FUNCTION_BLOCK FB_SlaveRobot
VAR
	// slave arms, responsible for arm kinematic and control
	m_slaveArms :ARRAY[1..g_sArmNum] OF FB_SlaveArm;
	
	// arm light control word
	m_lightCrlWord :ARRAY [1..4] OF UDINT;
	
	// arm state
	m_slaveArmState:ARRAY[1..g_sArmNum] OF E_SlaveArmState:=[g_sArmNum(E_SlaveArmState.SlaveArmState_Error)];
	m_lastSlaveArmState:ARRAY[1..g_sArmNum] OF E_SlaveArmState:=[g_sArmNum(E_SlaveArmState.SlaveArmState_Error)];
	m_nextSlaveArmState:ARRAY[1..g_sArmNum] OF E_SlaveArmState:=[g_sArmNum(E_SlaveArmState.SlaveArmState_Error)];
	
	// flag if panel and instrument mounted
	m_panelMountedFlag :ARRAY[1..g_sArmNum] OF BOOL :=[g_sArmNum(FALSE)];
	m_instrumentMountedFlag :ARRAY[1..g_sArmNum] OF BOOL :=[g_sArmNum(FALSE)];
	
	// all arm controller instance 
	m_armCtrlFactory :ARRAY[1..g_sArmNum,1..SlaveArmState_totalNum] OF I_SlaveArmCtrl;
	m_armError :ARRAY[1..g_sArmNum] OF FB_SlaveCtrlError;
	m_armInit :ARRAY[1..g_sArmNum] OF FB_SlaveCtrlInit;
	m_armSelfCheck :ARRAY[1..g_sArmNum] OF FB_SlaveCtrlSelfCheck;
	m_armStandBy :ARRAY[1..g_sArmNum] OF FB_SlaveCtrlStandBy;
	m_mountPanel :ARRAY[1..g_sArmNum] OF FB_SlaveCtrlMountPanel;
	m_panelReady :ARRAY[1..g_sArmNum] OF FB_SlaveCtrlPanelReady;
	m_mountInstru :ARRAY[1..g_sArmNum] OF FB_SlaveCtrlMountInstru;
	m_instruReady :ARRAY[1..g_sArmNum] OF FB_SlaveCtrlInstruReady;
	m_armMasterSlave :ARRAY[1..g_sArmNum] OF FB_SlaveCtrlMasterSlave;
	m_scopeReady :ARRAY[1..g_sArmNum] OF FB_SlaveCtrlScopeReady;
	m_armEndoscope :ARRAY[1..g_sArmNum] OF FB_SlaveCtrlEndoscope;
	m_armAdjust :ARRAY[1..g_sArmNum] OF FB_SlaveCtrlAdjust;
	m_armPackage :ARRAY[1..g_sArmNum] OF FB_SlaveCtrlPackage;
	m_armCart :ARRAY[1..g_sArmNum] OF FB_SlaveCtrlCart;
	m_armGraCali :ARRAY[1..g_sArmNum] OF FB_SlaveCtrlGraCali;
	m_armTest :ARRAY[1..g_sArmNum] OF FB_SlaveCtrlTest;
	m_instruRetract :ARRAY[1..g_sArmNum] OF FB_SlaveCtrlInstruRetract;
	m_instruInvasion :ARRAY[1..g_sArmNum] OF FB_SlaveCtrlInstruInvasion;
	m_armDisable :ARRAY[1..g_sArmNum] OF FB_SlaveCtrlDisable;
	m_instruCali :ARRAY[1..g_sArmNum] OF FB_SlaveCtrlInstruCali;
	m_scopeToggle :ARRAY[1..g_sArmNum] OF FB_SlaveCtrlScopeToggle;
	m_Performance :ARRAY[1..g_sArmNum] OF FB_SlaveCtrlPerformance;
	m_armStop :ARRAY[1..g_sArmNum] OF FB_SlaveCtrlStop;
	m_instruAutoTest :ARRAY[1..g_sArmNum] OF FB_SlaveCtrlInstruAutoTest;
	m_instruManualTest :ARRAY[1..g_sArmNum] OF FB_SlaveCtrlInstruManualTest;
	m_instruVerify :ARRAY[1..g_sArmNum] OF FB_SlaveCtrlInstruVerify;
	m_frictionTest :ARRAY[1..g_sArmNum] OF FB_SlaveCtrlFrictionTest;
	
	m_jnt5Rotate :ARRAY[1..g_sArmNum] OF FB_SlaveCtrlJnt5Rotate;
	
	// arm controller interface
	m_armCtrl :ARRAY[1..g_sArmNum] OF I_SlaveArmCtrl;
	m_armCtrlCmds :ARRAY[1..g_sArmNum] OF ST_SlaveArmCtrlCmds;
	m_motorGoHome: ARRAY[1..g_sArmNum] OF FB_SlaveCtrMotorGoHome;
	m_powerBoxCalibration: ARRAY[1..g_sArmNum] OF FB_SlaveCtrlPowerBoxCalibration;
	fbTonMotorGoHomeState: TON;
	fbTonPowerBoxCalibrationState: TON;
	m_endoscopeTest: ARRAY[1..g_sArmNum] OF FB_SlaveCtrlInstruEndoscopeTest;
	m_enableMode:BOOL;
END_VAR

METHOD PROTECTED controllerTransit : BOOL
VAR_INPUT
END_VAR
VAR
	i:int;
END_VAR
FOR i:=1 TO g_sArmNum DO 
	// Controller transit
	IF m_nextSlaveArmState[i]<> m_slaveArmState[i] THEN
		// reset current controller
		m_armCtrl[i].reset();
		
		// transit to new controller
		m_lastSlaveArmState[i]:=m_slaveArmState[i];
		m_slaveArmState[i]:=m_nextSlaveArmState[i];
		m_armCtrl[i]:=m_armCtrlFactory[i,m_slaveArmState[i]];
		
		// init next controller
		m_armCtrl[i].Init(m_slaveArms[i],m_armCtrlCmds[i]);
		m_slaveArms[i].updateCmds(m_armCtrlCmds[i]);
	END_IF
END_FOR
END_METHOD

METHOD PUBLIC Init : BOOL
VAR_INPUT
END_VAR
VAR
	i:INT;
END_VAR
FOR i:=1 TO g_sArmNum DO
	// arm init
	m_slaveArms[i].Init(i);
	m_slaveArmState[i]:=SlaveArmState_Init;
	m_lastSlaveArmState[i]:=SlaveArmState_Init;
	m_nextSlaveArmState[i]:=SlaveArmState_Init;
	
	// command init
	m_armCtrlCmds[i].m_jntEnableFlag := g_zeroVec8i;
	m_armCtrlCmds[i].m_jntOPMode := g_slaveAllPosMode;
	m_armCtrlCmds[i].m_cmdCartPose := m_slaveArms[i].curCartPose;
	m_armCtrlCmds[i].m_cmdCartTwist := g_zeroVec6d;
	m_armCtrlCmds[i].m_cmdJntPos := m_slaveArms[i].curJntPos;
	m_armCtrlCmds[i].m_cmdJntVel := g_zeroVec8d;
	m_armCtrlCmds[i].m_cmdJntAcc := g_zeroVec8d;
	m_armCtrlCmds[i].m_cmdJntTrq := g_zeroVec8d;
	
	// generate controller factory
	m_armCtrlFactory[i,SlaveArmState_Error] := m_armError[i];
	m_armCtrlFactory[i,SlaveArmState_Init] := m_armInit[i];
	m_armCtrlFactory[i,SlaveArmState_SelfCheck] := m_armSelfCheck[i];
	m_armCtrlFactory[i,SlaveArmState_Standby] := m_armStandBy[i];
	m_armCtrlFactory[i,SlaveArmState_MountPanel] := m_mountPanel[i];
	m_armCtrlFactory[i,SlaveArmState_PanelReady] := m_panelReady[i];
	m_armCtrlFactory[i,SlaveArmState_MountInstru] := m_mountInstru[i];
	m_armCtrlFactory[i,SlaveArmState_InstruReady] := m_instruReady[i];
	m_armCtrlFactory[i,SlaveArmState_MasterSlave] := m_armMasterSlave[i];
	m_armCtrlFactory[i,SlaveArmState_ScopeReady] := m_scopeReady[i];
	m_armCtrlFactory[i,SlaveArmState_EndoScope] := m_armEndoscope[i];
	m_armCtrlFactory[i,SlaveArmState_Adjust] := m_armAdjust[i];
	m_armCtrlFactory[i,SlaveArmState_Package] := m_armPackage[i];
	m_armCtrlFactory[i,SlaveArmState_Cart] := m_armCart[i];
	m_armCtrlFactory[i,SlaveArmState_GravityCali] := m_armGraCali[i];
	m_armCtrlFactory[i,SlaveArmState_Test] := m_armTest[i];
	m_armCtrlFactory[i,SlaveArmState_InstruRetract] := m_instruRetract[i];
	m_armCtrlFactory[i,SlaveArmState_InstruInvasion] := m_instruInvasion[i];
	m_armCtrlFactory[i,SlaveArmState_Disable] := m_armDisable[i];
	m_armCtrlFactory[i,SlaveArmState_InstruCali] := m_instruCali[i];
	m_armCtrlFactory[i,SlaveArmState_ScopeToggle] := m_scopeToggle[i];
	m_armCtrlFactory[i,SlaveArmState_Performance] := m_Performance[i];
	m_armCtrlFactory[i,SlaveArmState_Stop] := m_armStop[i];
	m_armCtrlFactory[i,SlaveArmState_InstruAutoTest] := m_instruAutoTest[i];
	m_armCtrlFactory[i,SlaveArmState_InstruManualTest] := m_instruManualTest[i];
	m_armCtrlFactory[i,SlaveArmState_InstruVerify] := m_instruVerify[i];
	m_armCtrlFactory[i,SlaveArmState_MotorGoHome] := m_motorGoHome[i];
	m_armCtrlFactory[i,SlaveArmState_PowerBoxCalibration] := m_powerBoxCalibration[i];
	m_armCtrlFactory[i,SlaveArmState_EndoscopeTest] := m_endoscopeTest[i];
	m_armCtrlFactory[i,SlaveArmState_FrictionTest] := m_frictionTest[i];
	
	m_armCtrlFactory[i,SlaveArmState_Jnt5Rotate] := m_jnt5Rotate[i];
	
	// assign controller
	m_armCtrl[i]:=m_armCtrlFactory[i,m_slaveArmState[i]];
	m_armCtrl[i].Init(m_slaveArms[i],m_armCtrlCmds[i]);
END_FOR
END_METHOD

METHOD PUBLIC run : BOOL
VAR_IN_OUT CONSTANT
	i_slaveInputDataPool:ST_SlaveInputDataPool;
END_VAR
VAR
	i:INT;
	nullScopePose :ST_Frame;
	nullSetupStatus:ST_SetupStatus;
	nullMasterStatus:ST_MasterStatus;
	
	
END_VAR
FOR i:=1 TO g_sArmNum DO
	// update dynamic data
	m_slaveArms[i].updateDyna(i_slaveInputDataPool.m_slaveDynaData);
								
	// update slave arm kinematics
	m_slaveArms[i].updateStatus();
END_FOR

//update arm light
updateArmLight(i_slaveInputDataPool);

// state machine transition
stateMachine(i_slaveInputDataPool);

// controller transition
controllerTransit();

FOR i:=1 TO g_sArmNum DO
	// null ptr check
	ASSERT(0 <> m_armCtrl[i]);
	
	// run controller
	m_armCtrl[i].run(nullScopePose, nullMasterStatus, nullSetupStatus,m_SlaveArms[i],m_armCtrlCmds[i]);

	// update commands to drivers
	m_slaveArms[i].updateCmds(m_armCtrlCmds[i]);

END_FOR
// ################# update insrument UI data #########################################
FOR i:=1 TO 5 DO 
	GVL_InstruTestUIVars.g_curInstruJntPos[i]:= m_slaveArms[1].curJntPos[i+3];
	GVL_InstruTestUIVars.g_curInstruJntCurrent[i]:= m_slaveArms[1].filtJntCurrent[i+3];
	GVL_InstruTestUIVars.g_instruZeroPos[i]:= m_slaveArms[1].instrument.onChipData.m_InstruPos[i];
END_FOR

FOR i:=1 TO 3 DO
		GVL_InstruTestUIVars.g_curInstruDHPos[i]:= m_slaveArms[1].curDHJntPos[i+3];
END_FOR

GVL_InstruTestUIVars.g_curGripAng := m_slaveArms[1].curGripAngle;
GVL_InstruTestUIVars.g_enabled := m_slaveArms[1].m_joints[6].isEnabled() ;
END_METHOD

// state machine check and transit 
METHOD PROTECTED stateMachine : BOOL
VAR_IN_OUT CONSTANT
		i_slavesInputDataPool:ST_SlaveInputDataPool;
END_VAR
VAR
	i,j:INT;
END_VAR
// check instrument state
FOR i:=1 TO g_sArmNum DO
	// statues check
	IF m_slaveArms[i].panelOn = FALSE THEN
		m_panelMountedFlag[i]:=FALSE;
	END_IF
	IF m_slaveArms[i].instruOn = FALSE THEN
		m_instrumentMountedFlag[i]:=FALSE;
	END_IF
END_FOR
// state machine transit
FOR i:=1 TO g_sArmNum DO
	CASE m_slaveArmState[i] OF
		// init
		SlaveArmState_Init:
			m_slaveArms[i].instrument.resetArmLED :=TRUE;
			// to standby
			IF m_armCtrl[i].isFinished  THEN
				m_nextSlaveArmState[i]:=SlaveArmState_Standby;
			END_IF
		
		//standby
		SlaveArmState_Standby:
			// to mount panel
			IF m_slaveArms[i].panelOn AND ((GVL_InstruTestUIVars.g_snappingSeparator AND NOT m_slaveArms[i].instruOn) OR  m_panelMountedFlag[i] )AND NOT GVL_InstruTestUIVars.g_powerBoxCalibration THEN 
				IF m_panelMountedFlag[i] THEN
					m_nextSlaveArmState[i]:=SlaveArmState_PanelReady;
				ELSE
					m_nextSlaveArmState[i]:=SlaveArmState_MountPanel;
				END_IF
			ELSIF GVL_InstruTestUIVars.g_goHome AND NOT m_slaveArms[i].instruOn THEN  
				GVL_InstruTestUIVars.g_beHomed:=FALSE;
				m_nextSlaveArmState[i]:=SlaveArmState_MotorGoHome;
			END_IF
			IF GVL_InstruTestUIVars.g_powerBoxCalibration THEN
				GVL_InstruTestUIVars.g_powerBoxCalibrationed:=FALSE;;
				IF m_slaveArms[i].panelOn THEN 
					m_nextSlaveArmState[i]:=SlaveArmState_PowerBoxCalibration;
				END_IF
			END_IF
		SlaveArmState_MotorGoHome:
			// to Standby
			IF m_armCtrl[i]. isFinished THEN
				m_nextSlaveArmState[i]:=SlaveArmState_Standby;
				GVL_InstruTestUIVars.g_beHomed:=TRUE;
			// to standby
			ELSIF fbTonMotorGoHomeState.Q THEN
				m_nextSlaveArmState[i]:=SlaveArmState_Standby;
			END_IF
		SlaveArmState_PowerBoxCalibration:
			IF m_armCtrl[i]. isFinished THEN
				GVL_InstruTestUIVars.g_powerBoxCalibration:=FALSE;
				GVL_InstruTestUIVars.g_powerBoxCalibrationed:=TRUE;
				FOR j:=4 TO g_sJntNum DO
					GVL_InstruTestUIVars.g_powerBoxCalibrationPos[i,j]:=SlaveArmControl.m_slaveRobot.m_slaveArms[i].m_joints[j].m_motorInputs.m_linkEncoder;
				END_FOR
				GVL_SlaveJointEncoderCaliData.g_caliLinkEncoder:=GVL_InstruTestUIVars.g_powerBoxCalibrationPos;
				IF NOT m_slaveArms[i].panelOn THEN
					GVL_InstruTestUIVars.g_powerBoxCalibrationFlag:=FALSE;
					m_nextSlaveArmState[i]:=SlaveArmState_Standby;;
					m_slaveArms[i].setSaveCaliLinkEncoder();
				END_IF
			// to standby
			ELSIF fbTonPowerBoxCalibrationState.Q AND NOT m_slaveArms[i].panelOn THEN
				m_nextSlaveArmState[i]:=SlaveArmState_Standby;
			END_IF
		//mount panel
		SlaveArmState_MountPanel:
			// to panel ready
			IF m_armCtrl[i]. isFinished THEN
				m_nextSlaveArmState[i]:=SlaveArmState_PanelReady;
				m_panelMountedFlag[i] :=TRUE;
				
			// to standby
			ELSIF NOT(m_slaveArms[i].panelOn) THEN
				m_nextSlaveArmState[i]:=SlaveArmState_Standby;
			END_IF
		
		//panel ready
		SlaveArmState_PanelReady:
			// to standby
			IF NOT(m_slaveArms[i].panelOn) THEN
				m_nextSlaveArmState[i]:=SlaveArmState_Standby;
			
			// to instrument caliberation
			ELSIF GVL_InstruTestUIVars.g_instruCaliFlag THEN
				m_nextSlaveArmState[i] := SlaveArmState_InstruCali;
			ELSIF (GVL_InstruTestUIVars.g_instrumentAutoSnapping OR m_instrumentMountedFlag[i]) AND m_slaveArms[i].instruOn   THEN
				IF m_instrumentMountedFlag[i] THEN
					// to scope ready
					IF  InstruType_endoscope = m_slaveArms[i].instrument.m_instruType AND m_slaveArms[i].instruReady() THEN 
						m_nextSlaveArmState[i]:=SlaveArmState_ScopeReady;
					// to instrument ready
					ELSE
						m_nextSlaveArmState[i]:=SlaveArmState_InstruReady;
					END_IF
				// to mount instrument/endoscope
				ELSE
					m_nextSlaveArmState[i]:=SlaveArmState_MountInstru;
				END_IF
			END_IF
			
		//mount instrument
		SlaveArmState_MountInstru:
			// to panel ready
			IF NOT(m_slaveArms[i].instruOn)  THEN
				m_nextSlaveArmState[i]:=SlaveArmState_PanelReady;
			ELSIF m_armCtrl[i].isFinished THEN
				m_instrumentMountedFlag[i] :=TRUE;
				m_nextSlaveArmState[i]:=SlaveArmState_PanelReady;
				
			END_IF
		
		// instrument ready
		SlaveArmState_InstruReady:
			// to instrument standby
			IF  NOT(m_slaveArms[i].instruOn)  THEN
				m_nextSlaveArmState[i]:=SlaveArmState_Standby;
				GVL_InstruTestUIVars.g_readRFIDFlag:=FALSE;
			// to instrument caliberation
			ELSIF GVL_InstruTestUIVars.g_instruCaliFlag THEN
				m_nextSlaveArmState[i] := SlaveArmState_InstruCali;
				
			// to instrument auto test
			ELSIF GVL_InstruTestUIVars.g_instruAutoTestFlag THEN
				m_nextSlaveArmState[i] := SlaveArmState_InstruAutoTest;
				
			// to instrument manual test
			ELSIF GVL_InstruTestUIVars.g_instruManualTestFlag THEN
				m_nextSlaveArmState[i] := SlaveArmState_InstruManualTest;
				
			// to instrument verify
			ELSIF GVL_InstruTestUIVars.g_instruVerifyFlag THEN
				m_nextSlaveArmState[i] := SlaveArmState_InstruVerify;
				
			// to instrument verify
			ELSIF GVL_InstruTestUIVars.g_endoscopeTest THEN
				m_nextSlaveArmState[i] := SlaveArmState_EndoscopeTest;
				
			//to friction Test
			ELSIF GVL_InstruTestUIVars.g_instruFrictionTest THEN
				m_nextSlaveArmState[i] := SlaveArmState_FrictionTest;
			END_IF
			
		//instrument caliberation
		SlaveArmState_InstruCali:
			// to standby
			IF  NOT(GVL_InstruTestUIVars.g_instruCaliFlag)  THEN
				m_nextSlaveArmState[i]:=SlaveArmState_Standby;
			END_IF
			
		//instrument auto test
		SlaveArmState_InstruAutoTest:
			// to stop
			IF  NOT( m_slaveArms[1].instruOn) OR NOT(GVL_InstruTestUIVars.g_instruAutoTestFlag)  THEN
				m_nextSlaveArmState[i]:=SlaveArmState_Stop;
				GVL_InstruTestUIVars.g_readRFIDFlag:=FALSE;
				m_armStop[i].setInstruBacklash(m_instruAutoTest[i].InstruBacklash);
			END_IF
			IF m_armCtrl[i].isFinished THEN
				GVL_InstruTestUIVars.g_instruAutoTestFlag:=FALSE;
			END_IF
		//instrument manual test
		SlaveArmState_InstruManualTest:
			// to stop
			IF  NOT( m_slaveArms[1].instruOn) OR NOT(GVL_InstruTestUIVars.g_instruManualTestFlag)  THEN
				m_nextSlaveArmState[i]:=SlaveArmState_Stop;
				m_armStop[i].setInstruBacklash(m_instruManualTest[i].InstruBacklash);
				GVL_InstruTestUIVars.g_readRFIDFlag:=FALSE;
			END_IF
			
		//instrument verify
		SlaveArmState_InstruVerify:
			// to stop
			IF  NOT( m_slaveArms[1].instruOn) OR NOT(GVL_InstruTestUIVars.g_instruVerifyFlag)  THEN
				m_nextSlaveArmState[i]:=SlaveArmState_Stop;
				GVL_InstruTestUIVars.g_readRFIDFlag:=FALSE;
				m_armStop[i].setInstruBacklash(m_instruVerify[i].InstruBacklash);
			END_IF
			IF m_armCtrl[i].isFinished THEN
				GVL_InstruTestUIVars.g_instruVerifyFlag:=FALSE;
			END_IF
			
		//arm stop
		SlaveArmState_Stop:
			// to standby
			IF  m_armCtrl[i].isFinished THEN
				m_nextSlaveArmState[i]:=SlaveArmState_Standby;
			END_IF
			
		SlaveArmState_Disable:
			// to init
			IF  NOT GVL_InstruTestUIVars.g_powerOn  THEN
				m_nextSlaveArmState[i]:=SlaveArmState_Init;
			END_IF
		    IF  NOT( m_slaveArms[1].instruOn) THEN
				m_nextSlaveArmState[i]:=SlaveArmState_Init;
			END_IF
			
		SlaveArmState_EndoscopeTest:
			IF  NOT( m_slaveArms[1].instruOn) OR NOT(GVL_InstruTestUIVars.g_endoscopeTest)  THEN
				m_nextSlaveArmState[i]:=SlaveArmState_Stop;
			END_IF
			
		SlaveArmState_FrictionTest:
			// to stop
			IF  NOT( m_slaveArms[1].instruOn) OR m_armCtrl[i].isFinished OR NOT GVL_InstruTestUIVars.g_instruFrictionTest  THEN
				m_nextSlaveArmState[i]:=SlaveArmState_Standby;
			END_IF	
		
		SlaveArmState_Jnt5Rotate:
			// to standby
			IF  m_armCtrl[i].isFinished THEN
				m_nextSlaveArmState[i]:=SlaveArmState_Standby;
			END_IF
	END_CASE
	
	IF NOT m_slaveArms[i].instruOn THEN
		GVL_InstruTestUIVars.g_instruCaliState:=FALSE;
	END_IF
	IF GVL_InstruTestUIVars.g_powerOn THEN 
		m_nextSlaveArmState[i]:=SlaveArmState_Disable;
	END_IF
	IF GVL_InstruTestUIVars.g_motorStops THEN 
		GVL_InstruTestUIVars.g_motorStops:=FALSE;
		m_nextSlaveArmState[i]:=SlaveArmState_Stop;
	END_IF
	
	
	IF GVL_InstruTestUIVars.g_jnt5RotateFlag THEN
		m_nextSlaveArmState[i]:=SlaveArmState_Jnt5Rotate;
		GVL_InstruTestUIVars.g_jnt5RotateFlag:=FALSE;
	END_IF
	
	IF m_slaveArmState[i]<>SlaveArmState_PowerBoxCalibration AND m_slaveArmState[i]<>SlaveArmState_Standby THEN
		GVL_InstruTestUIVars.g_powerBoxCalibration:=FALSE;
	END_IF
	IF m_slaveArmState[i]<>SlaveArmState_MotorGoHome AND m_slaveArmState[i]<>SlaveArmState_Standby THEN
		GVL_InstruTestUIVars.g_beHomed:=FALSE;
	END_IF
	
	
GVL_InstruTestUIVars.g_stateMachine:=m_slaveArmState[i];
	IF GVL_InstruTestUIVars.g_manualPowerBoxCalibration THEN
		FOR j:=4 TO g_sJntNum DO
			GVL_InstruTestUIVars.g_powerBoxCalibrationPos[i,j]:=SlaveArmControl.m_slaveRobot.m_slaveArms[i].m_joints[j].m_motorInputs.m_linkEncoder;
		END_FOR
		GVL_SlaveJointEncoderCaliData.g_caliLinkEncoder:=GVL_InstruTestUIVars.g_powerBoxCalibrationPos;
		GVL_InstruTestUIVars.g_manualPowerBoxCalibration:=FALSE;
		GVL_InstruTestUIVars.g_powerBoxCalibrationFlag:=FALSE;
		m_slaveArms[i].setSaveCaliLinkEncoder();
	END_IF
END_FOR


m_enableMode:=TRUE;
GVL_InstruTestUIVars.g_logOutEnable:=GVL_InstruTestUIVars.g_stateMachine<>SlaveArmState_InstruAutoTest;
GVL_InstruTestUIVars.g_snappingSeparatoring:=GVL_InstruTestUIVars.g_stateMachine=SlaveArmState_MountPanel;
GVL_InstruTestUIVars.g_instruAutoSnapping:=GVL_InstruTestUIVars.g_stateMachine=SlaveArmState_MountInstru;
GVL_InstruTestUIVars.g_instruCalibrationing:=m_instruCali[1].getState AND GVL_InstruTestUIVars.g_stateMachine=SlaveArmState_InstruCali;
GVL_MES.g_autoTestMode:=m_instruAutoTest[1].getTestMode;
GVL_InstruTestUIVars.g_forceBipolarModeAllowed := InstruType_ForceBipolar = m_slaveArms[1].instrument.instruTypeInfo.m_InstruID;
GVL_InstruTestUIVars.g_instruFrictionTestAllowed := m_slaveArms[1].instrument.onChipData.m_InstruReadSucceed AND m_instrumentMountedFlag[1];
GVL_InstruTestUIVars.g_testEnable:=m_slaveArms[1].instrument.onChipData.m_InstruReadSucceed AND m_instrumentMountedFlag[1];
IF NOT GVL_InstruTestUIVars.g_testEnable THEN
	GVL_InstruTestUIVars.g_instruAutoTestFlag:=FALSE;
	GVL_InstruTestUIVars.g_instruManualTestFlag:=FALSE;
	GVL_InstruTestUIVars.g_instruVerifyFlag:=FALSE;
END_IF
GVL_InstruTestUIVars.g_standbyEnable:=GVL_InstruTestUIVars.g_stateMachine=SlaveArmState_Standby AND NOT m_slaveArms[1].panelOn;
END_METHOD

METHOD updateArmLight : BOOL
VAR_INPUT
	i_slaveInputDataPool:ST_SlaveInputDataPool;
END_VAR

VAR
	i : INT;
END_VAR
//*******************机械臂与动力盒上的灯光写入********************
//不可恢复性故障-----红色常亮
//可恢复故障----琥珀色-先闪烁5s、再进行常亮
//正处于器械控制或者端口控制状态-----蓝色闪烁
//该手术臂正在执行一项需要用户短时间等待的活动、例如器械卡接----蓝色-脉动闪烁
//工具更换引导正在进行中-----绿色闪烁
//未通电、已禁用、已收起----------关
//系统正常运行-----蓝色常亮
//灯光颜色--0-灯灭、1蓝灯常亮、2蓝灯闪烁、3琥珀色闪烁、4红灯闪烁、5绿灯常亮、6绿灯闪烁、7红灯常亮、8琥珀色常亮、9蓝灯脉动式闪烁

FOR i := 1 TO g_sArmNum BY 1 DO
	IF m_slaveArmState[i] = SlaveArmState_Error THEN
		m_lightCrlWord[i] := ArmLight_AmberBlink;
	ELSIF m_slaveArmState[i] = SlaveArmState_MountPanel OR m_slaveArmState[i] = SlaveArmState_MountInstru THEN
		m_lightCrlWord[i] := ArmLight_BluePulse;
	ELSIF m_slaveArmState[i] = SlaveArmState_InstruRetract OR m_slaveArmState[i] = SlaveArmState_Adjust THEN
		m_lightCrlWord[i] := ArmLight_BlueBlink;
	ELSIF m_slaveArmState[i] = SlaveArmState_InstruInvasion THEN
		m_lightCrlWord[i] := ArmLight_GreenBlink;
	ELSIF m_slaveArmState[i] = SlaveArmState_Disable THEN
		m_lightCrlWord[i] := ArmLight_Off;
	ELSE
		m_lightCrlWord[i] := ArmLight_BlueOn;
	END_IF

	m_slaveArms[i].checkLight(m_lightCrlWord[i]);
END_FOR
END_METHOD

END_FUNCTION_BLOCK

(* stored: Version 1.1.0.1, ProductVersion 3.1.4024.11
   POU FB_SlaveRobot: Id {8cbdb2ba-9735-46e3-8cbc-296330acc8cc}, SpecialFunc None
   Method controllerTransit: Id {8f288ee3-c1dd-4604-a493-d121fbcd6b66}
   Method Init: Id {610a17f3-34c5-4e3c-bbbc-19f9c2f46946}
   Method run: Id {ed6f787a-4dc0-4602-b386-92a3c3880a23}
   Method stateMachine: Id {b9cc8560-9309-49e3-93b5-28cb02b4f5cc}
   Method updateArmLight: Id {0d4d98a3-ae97-4bc5-8d05-6e3f5cc1e792} *)
